SYSTEM testProject
  (* Version 1.0, 2025-07-11, Дмитрий *)
  APPLICATION testProjectApp
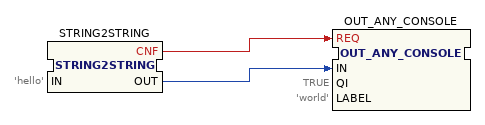
    FBS
      STRING2STRING : STRING2STRING(IN := 'hello');
      OUT_ANY_CONSOLE : OUT_ANY_CONSOLE(QI := TRUE, LABEL := 'world');
    END_FBS
    EVENT_CONNECTIONS
      STRING2STRING.CNF TO OUT_ANY_CONSOLE.REQ;
    END_CONNECTIONS
    DATA_CONNECTIONS
      STRING2STRING.OUT TO OUT_ANY_CONSOLE.IN;
    END_CONNECTIONS
  END_APPLICATION
  DEVICE FORTE_PC : FORTE_PC(MGR_ID := "localhost:61499")
    {SET_ATTRIBUTE(Profile, HOLOBLOC)} (* device profile *)
    RESOURCE EMB_RES : EMB_RES
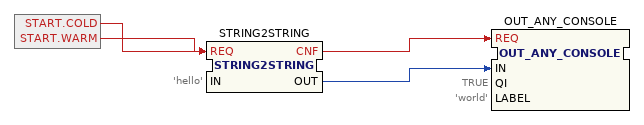
      FBS
        STRING2STRING : STRING2STRING(IN := 'hello');
        OUT_ANY_CONSOLE : OUT_ANY_CONSOLE(QI := TRUE, LABEL := 'world');
      END_FBS
      EVENT_CONNECTIONS
        STRING2STRING.CNF TO OUT_ANY_CONSOLE.REQ;
        START.COLD TO STRING2STRING.REQ;
        START.WARM TO STRING2STRING.REQ;
      END_CONNECTIONS
      DATA_CONNECTIONS
        STRING2STRING.OUT TO OUT_ANY_CONSOLE.IN;
      END_CONNECTIONS
    END_RESOURCE
  END_DEVICE
  MAPPINGS
    testProjectApp.STRING2STRING ON FORTE_PC.EMB_RES.STRING2STRING;
    testProjectApp.OUT_ANY_CONSOLE ON FORTE_PC.EMB_RES.OUT_ANY_CONSOLE;
  END_MAPPINGS
  SEGMENTS
    Ethernet : Ethernet;
  END_SEGMENTS
  LINKS
    FORTE_PC => Ethernet;
  END_LINKS
END_SYSTEM
